FUNCTION_BLOCK ButtonCheck
VAR
	Start 	: BOOL;
	EStop 	: BOOL;
	Reset	: BOOL;
	
END_VAR

METHOD mEStop : BOOL
VAR_INPUT
END_VAR
//pEStop := Buttons.EStop := TRUE; (Faulty)
pEStop := TRUE;
END_METHOD

METHOD mReset : BOOL
VAR_INPUT
END_VAR
pReset := TRUE;
END_METHOD

METHOD mStart : BOOL
VAR_INPUT
END_VAR
pStart := TRUE;
END_METHOD

PROPERTY pEStop : BOOL
GET
pEStop := EStop;
END_GET
SET
EStop := pEStop;
END_SET
END_PROPERTY

PROPERTY pReset : BOOL
GET
pReset := Reset;
END_GET
SET
Reset := pReset;
END_SET
END_PROPERTY

PROPERTY pStart : BOOL
GET
pStart := Start;
END_GET
SET
Start := pStart;
END_SET
END_PROPERTY

END_FUNCTION_BLOCK

(* stored: Version 1.1.0.1, ProductVersion 3.1.4024.9
   POU ButtonCheck: Id {1fe9154a-ebe7-4454-8b4c-d5c4945e70fc}, SpecialFunc None
   Method mEStop: Id {ceebe3ee-6bfd-406e-810b-501ff2ef2575}
   Method mReset: Id {18331239-0c7b-4c32-876a-64c2c13528ff}
   Method mStart: Id {21485928-264e-4c71-ae22-cb353a66a36d}
   Property pEStop: Id {69fb0f0b-dbe5-44bf-a64a-58ab8276e962}
   Get Get: Id {453c2299-fe14-447e-bcf4-0e6c756b8bb6}
   Set Set: Id {683bb7c9-b33d-4e17-be7e-394d73ccd1a6}
   Property pReset: Id {18a5e3b3-bc9c-432b-af97-893024fd5015}
   Get Get: Id {1c0bba4a-a90e-4839-a851-3b5932de4e29}
   Set Set: Id {58c40a54-1d5e-4413-bfe5-7b3017ee4367}
   Property pStart: Id {50607114-1ffb-470c-ba29-dd77a0a6669b}
   Get Get: Id {8ebe71c2-c921-4e77-b0dc-bd59403e5e4c}
   Set Set: Id {820c2e4c-585a-469a-bd89-22549140aae6} *)
